// TIA Portal V18 export
FUNCTION "calc_speeds_from_mechanics_1StepperMotor" : Void   // FC33, FBD
{ S7_Optimized_Access := 'TRUE' }
VERSION : 0.1
// stored: AutoNumber true, IsIECCheckEnabled false, SetENOAutomatically false, UDAEnableTagReadback false
   VAR_INPUT
      Vabsmax_deg_per_s : Real;
   END_VAR
   VAR_OUTPUT
      ER_params : Bool;
   END_VAR
   VAR_IN_OUT
      para : "typeMotPara";
   END_VAR
   VAR_TEMP
      counts_per_deg : Real;
      t_acceleration_s : Real;
      "a" : Real;
      v_abs_max : Real;
      t_mx : Real;
      v_min_viable : Real;
      dist_stop : Real;
      dist_auto_done : Real;
      K_min : Real;
      K_min_dist : Real;
      dist_absMax : Real;
   END_VAR
BEGIN

REGION Network 1 (SCL)
   #v_abs_max := #Vabsmax_deg_per_s;
   #t_acceleration_s := #para.t_acc_50Hz_USER;

   #K_min := 0.5 / 50.0;
   #v_min_viable := #v_abs_max * #K_min;

   #t_mx := #t_acceleration_s;
   #ER_params := #t_acceleration_s = 0 OR #v_abs_max = 0 OR #t_mx =0 ;
   IF NOT #ER_params THEN
       #a := #v_abs_max / #t_mx;
       #dist_absMax := #a * #t_mx * #t_mx / 2 + #v_min_viable * #t_mx;
   ELSE
       #a := 0;
        #dist_absMax := 999;
   END_IF;
   #K_min_dist :=0.5/ 50.0 ;//#K_min * 0.8;
   #dist_stop := #dist_absMax * #K_min_dist;
   #dist_auto_done := #dist_stop * 1.2;
END_REGION

REGION Network 2 (SCL)
   //#para.dist_absMax_LOGIC := #dist_fast;
   #para.dist_stop_USER := #dist_stop;
   #para.dist_auto_done_LOGIC := #dist_auto_done;
   //#para.dist_auto_maxCor_LOGIC := 0.1 * #para.dist_absMax_LOGIC;
   #para.v_absoluteMax_LOGIC := #v_abs_max;
   #para.v_crawl_USER := #v_min_viable;
   //#para.v_auto_maxCor_LOGIC := 0.1 * #para.v_absoluteMax_LOGIC;
END_REGION
END_FUNCTION
